{attribute 'GeneratedUsingTerminal: EM7004-0000-0016'}
{attribute addProperty BoxType "EM7004-0000-0016"}
{attribute addProperty Id "Latch_extern_validAT %I*BOOL1Set_counter_doneAT %I*BOOL1Status_of_input_AAT %I*BOOL1Status_of_input_BAT %I*BOOL1Status_of_input_gateAT %I*BOOL1Status_of_extern_latchAT %I*BOOL1TxPDO_ToggleAT %I*BOOL1Counter_valueAT %I*UINT2Latch_valueAT %I*UINT2"}
{attribute addProperty CRC "1802475527"}
{attribute addProperty Size "11"}
TYPE ENC_Inputs_Channel_6B6F9807 :
STRUCT
	{attribute addProperty Name "Latch_extern_valid"}
	Latch_extern_valid AT %I* : BOOL;
	{attribute addProperty Name "Set_counter_done"}
	Set_counter_done AT %I* : BOOL;
	{attribute addProperty Name "Status_of_input_A"}
	Status_of_input_A AT %I* : BOOL;
	{attribute addProperty Name "Status_of_input_B"}
	Status_of_input_B AT %I* : BOOL;
	{attribute addProperty Name "Status_of_input_gate"}
	Status_of_input_gate AT %I* : BOOL;
	{attribute addProperty Name "Status_of_extern_latch"}
	Status_of_extern_latch AT %I* : BOOL;
	{attribute addProperty Name "TxPDO_Toggle"}
	TxPDO_Toggle AT %I* : BOOL;
	{attribute addProperty Name "Counter_value"}
	Counter_value AT %I* : UINT;
	{attribute addProperty Name "Latch_value"}
	Latch_value AT %I* : UINT;
END_STRUCT
END_TYPE

(* stored: Version 1.2.0.0, ProductVersion 3.1.4024.9
   DUT ENC_Inputs_Channel_6B6F9807: Id {4155d09d-1053-4d70-8412-571f9aa4cfc7} *)
